{region '#Template'}
	{attribute 'Version' := '5.0.0.0'}
	{attribute 'Tags' := '"LCID": "1031", "Text": "General, Cabinet, Control cabinet, Acknowledgement"'}
	{attribute 'Tags' := '"LCID": "1033", "Text": "General, Cabinet, Control cabinet, Acknowledgement"'}
	{attribute 'Using' := '"Type": "Template", "URI": "EC_ID"'}
	{attribute 'Description' := '"LCID": "1031", "Text": "Schaltschrank Quittierung"'}
	{attribute 'Description' := '"LCID": "1033", "Text": "Control cabinet acknowledgement"'}
{endregion}
FUNCTION_BLOCK FB_BA_ControlCabinetBasicExt EXTENDS FB_BA_VIEW
VAR_INPUT
END_VAR
VAR_INPUT CONSTANT
	LampFault				: FB_BA_ActuatorCmd;		
	AckButton				: FB_BA_CombinationBI_BV;													
	EventObserver			: FB_BA_EventObserver;
END_VAR
VAR				
	bHasEvents				: BOOL;
	bHasUnackEvent			: BOOL;
	bTrigRstSwi				: BOOL;
	bTrigRstButton			: BOOL;	
END_VAR
VAR // added by the converter: edge detectors and wires of the graphical bodies
    _s1 : ST_BA_Binary;
END_VAR

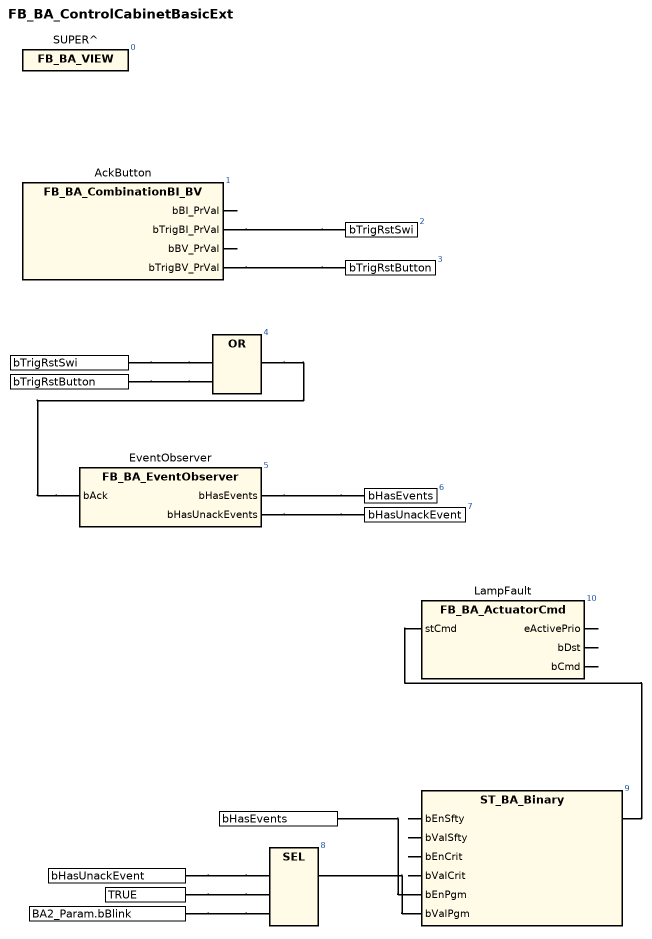
SUPER^(); // FB_BA_VIEW
AckButton(); // FB_BA_CombinationBI_BV
bTrigRstSwi := AckButton.bTrigBI_PrVal;
bTrigRstButton := AckButton.bTrigBV_PrVal;
EventObserver(bAck := bTrigRstSwi OR bTrigRstButton); // FB_BA_EventObserver
bHasEvents := EventObserver.bHasEvents;
bHasUnackEvent := EventObserver.bHasUnackEvents;
// compose _s1 : ST_BA_Binary
_s1.bEnPgm := bHasEvents;
_s1.bValPgm := SEL(bHasUnackEvent, TRUE, BA2_Param.bBlink);
LampFault(stCmd := _s1); // FB_BA_ActuatorCmd

METHOD FB_init : BOOL
VAR_INPUT
	bInitRetains : BOOL; // if TRUE, the retain variables are initialized (warm start / cold start)
	bInCopyCode : BOOL;  // if TRUE, the instance afterwards gets moved into the copy code (online change)
END_VAR
LampFault.iParent							:= THIS^;
LampFault.iLabel							:= LblCtl_EventIndicationLamp;
//LampFault.eDPADMode						:= E_BA_DPADMode.eInclude;	
LampFault.Cmd.iLabel						:= LblFun_SwitchingCommand;		
LampFault.Cmd.ePolarity						:= E_BA_Polarity.eNormal;
LampFault.Cmd.sActiveText 					:= txtEvent_On;
LampFault.Cmd.sInactiveText 				:= txtEvent_Off;
LampFault.Cmd.nEventClassID					:= EC_ID.NC40;
LampFault.Cmd.aEventTransitionText[1]		:= txtEvent_Disturb;
LampFault.Cmd.aEventTransitionText[2]		:= txtEvent_None;
LampFault.Cmd.aEventTransitionText[3]		:= txtEvent_Normal;
LampFault.Cmd.bEventDetectionEnable			:= FALSE;
LampFault.Cmd.eEnPlantLock					:= E_BA_LockPriority.eNoLock;	

AckButton.iParent							:= THIS^;
AckButton.iLabel							:= LblCtl_Acknowledge;				
//AckButton.eDPADMode						:= E_BA_DPADMode.eInclude;
AckButton.Input.iLabel						:= LblCtl_ButtonLocalAcknowledgement;																										
AckButton.Input.ePolarity					:= E_BA_Polarity.eNormal;
AckButton.Input.bEventDetectionEnable		:= FALSE;
AckButton.Value.eToggleMode 				:= E_BA_ToggleMode.ePushButton;					

EventObserver.Parent						:= XBA_Globals.Top;
END_METHOD

END_FUNCTION_BLOCK

(* stored: Version 1.1.0.1, ProductVersion 3.1.4024.12
   POU FB_BA_ControlCabinetBasicExt: Id {a8bde42e-1bb9-4575-ab5f-a7759126a215}, SpecialFunc None
   Method FB_init: Id {602a88ff-269d-409b-8938-c22fa40d1460} *)
